FUNCTION F_RoundToClosest : UDINT
VAR_INPUT
	valueToBeRounded 			: UDINT;
	increment 					: UDINT;
	upperLimit 					: UDINT;
END_VAR
VAR
	valueDividedByIncrement		: UDINT;
END_VAR

valueDividedByIncrement := valueToBeRounded/increment;
IF valueToBeRounded MOD increment <> 0 THEN
	F_RoundToClosest := valueDividedByIncrement * increment + increment;
ELSE
	F_RoundToClosest := valueToBeRounded;
END_IF
IF F_RoundToClosest > upperLimit THEN
	F_RoundToClosest := upperLimit;
END_IF

END_FUNCTION

(* stored: Version 1.1.0.1, ProductVersion 3.1.4024.9
   POU F_RoundToClosest: Id {7f11ef65-8aa7-47e2-b8fb-aca6037dab01}, SpecialFunc None *)
